{attribute 'qualified_only'}
VAR_GLOBAL
	Test :BOOL;
	Data :ARRAY[0..100] OF INT;
	DAtatekst : string[255];
END_VAR

(* stored: Version 1.1.0.1, ProductVersion 3.1.4024.11
   GVL GVLDataproces: Id {999d4de7-4d73-43e9-b7a7-8d924654cb84} *)
